// Mitsubishi GX Works2 project: Test1   PLC: FX3U/FX3UC

PROGRAM MAIN
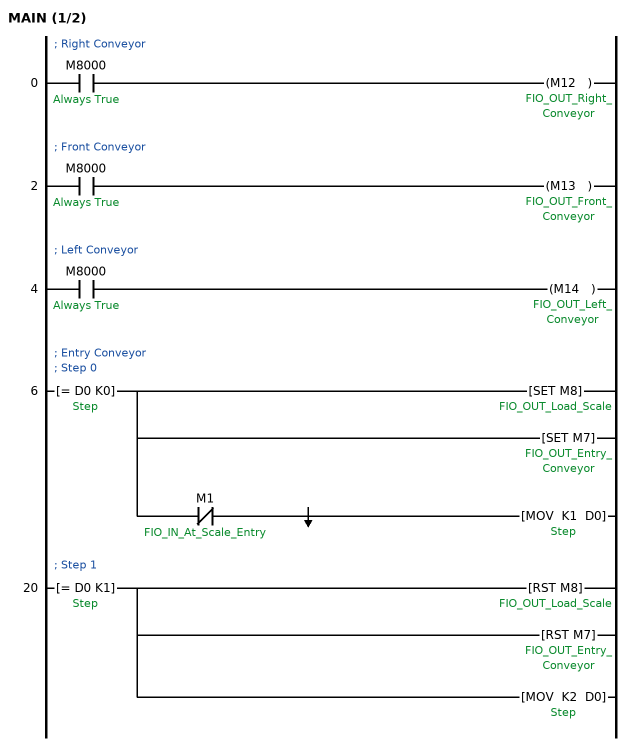
; Right Conveyor
0     LD      M8000  ; Always True
      OUT     M12  ; FIO_OUT_Right_Conveyor
; Front Conveyor
2     LD      M8000  ; Always True
      OUT     M13  ; FIO_OUT_Front_Conveyor
; Left Conveyor
4     LD      M8000  ; Always True
      OUT     M14  ; FIO_OUT_Left_Conveyor
; Entry Conveyor
; Step 0
6     LD=     D0 K0  ; Step
      SET     M8  ; FIO_OUT_Load_Scale
      SET     M7  ; FIO_OUT_Entry_Conveyor
      ANI     M1  ; FIO_IN_At_Scale_Entry
      MEF
      MOV     K1 D0
; Step 1
20    LD=     D0 K1  ; Step
      RST     M8  ; FIO_OUT_Load_Scale
      RST     M7  ; FIO_OUT_Entry_Conveyor
      MOV     K2 D0
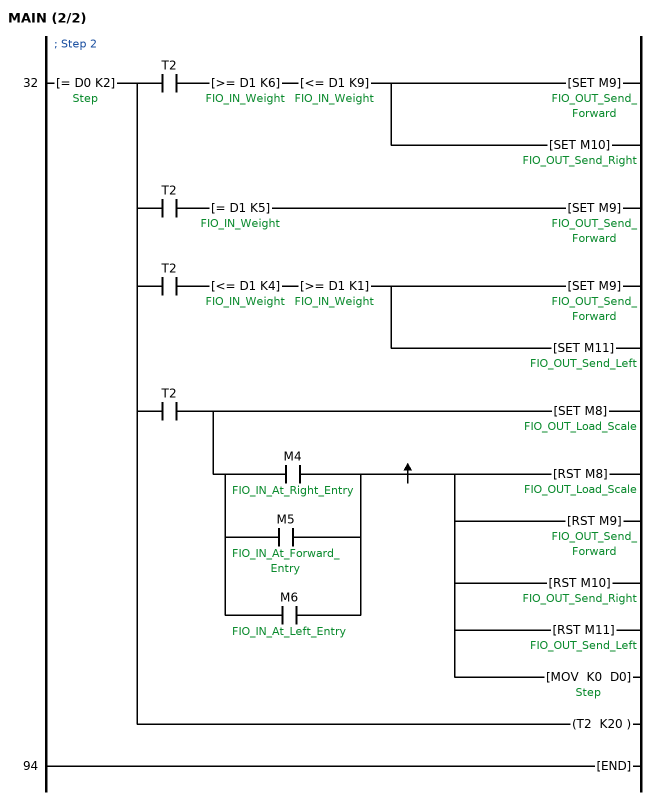
; Step 2
32    LD=     D0 K2  ; Step
      MPS
      AND     T2
      AND>=   D1 K6  ; FIO_IN_Weight
      AND<=   D1 K9  ; FIO_IN_Weight
      SET     M9  ; FIO_OUT_Send_Forward
      SET     M10  ; FIO_OUT_Send_Right
      MRD
      AND     T2
      AND=    D1 K5  ; FIO_IN_Weight
      SET     M9  ; FIO_OUT_Send_Forward
      MRD
      AND     T2
      AND<=   D1 K4  ; FIO_IN_Weight
      AND>=   D1 K1  ; FIO_IN_Weight
      SET     M9  ; FIO_OUT_Send_Forward
      SET     M11  ; FIO_OUT_Send_Left
      MRD
      AND     T2
      SET     M8  ; FIO_OUT_Load_Scale
      LD      M4  ; FIO_IN_At_Right_Entry
      OR      M5  ; FIO_IN_At_Forward_Entry
      OR      M6  ; FIO_IN_At_Left_Entry
      ANB
      MEP
      RST     M8  ; FIO_OUT_Load_Scale
      RST     M9  ; FIO_OUT_Send_Forward
      RST     M10  ; FIO_OUT_Send_Right
      RST     M11  ; FIO_OUT_Send_Left
      MOV     K0 D0
      MPP
      OUT     T2 K20
94    END
END_PROGRAM

// device comments not shown above
M2  ; FIO_IN_At_Scale
M3  ; FIO_IN_At_Scale_Exit
M15  ; FIO_OUT_Back_Ward
M16  ; FIO_OUT_Rescale
D2  ; Stored_Weight
